SYSTEM dets
  (* Version 1.0, 2023-01-24, obotnar *)
  APPLICATION detsApp
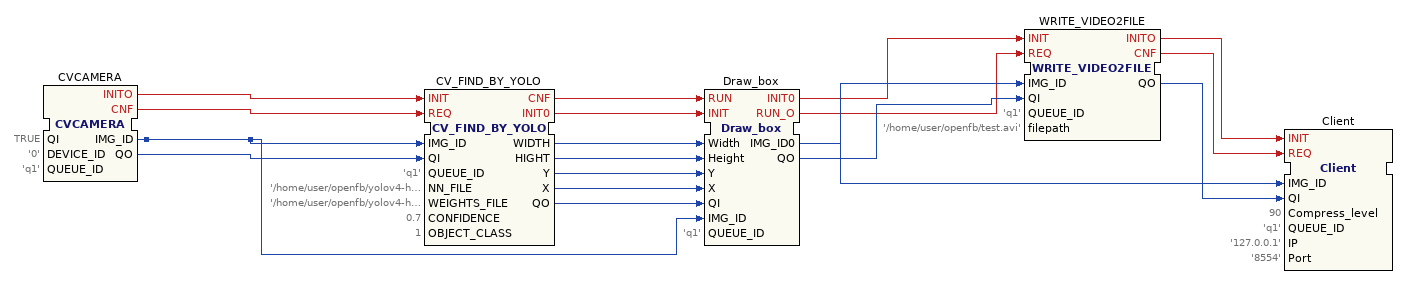
    FBS
      CV_FIND_BY_YOLO : CV_FIND_BY_YOLO(QUEUE_ID := 'q1', NN_FILE := '/home/user/openfb/yolov4-head-tiny-416.cfg', WEIGHTS_FILE := '/home/user/openfb/yolov4-head-tiny-416.weights', CONFIDENCE := 0.7, OBJECT_CLASS := 1);
      Draw_box : Draw_box(QUEUE_ID := 'q1');
      WRITE_VIDEO2FILE : WRITE_VIDEO2FILE(QUEUE_ID := 'q1', filepath := '/home/user/openfb/test.avi');
      Client : Client(Compress_level := 90, QUEUE_ID := 'q1', IP := '127.0.0.1', Port := '8554');
      CVCAMERA : CVCAMERA(QI := TRUE, DEVICE_ID := '0', QUEUE_ID := 'q1');
    END_FBS
    EVENT_CONNECTIONS
      CV_FIND_BY_YOLO.CNF TO Draw_box.RUN;
      CV_FIND_BY_YOLO.INIT0 TO Draw_box.INIT;
      Draw_box.INIT0 TO WRITE_VIDEO2FILE.INIT;
      Draw_box.RUN_O TO WRITE_VIDEO2FILE.REQ;
      WRITE_VIDEO2FILE.INITO TO Client.INIT;
      WRITE_VIDEO2FILE.CNF TO Client.REQ;
      CVCAMERA.INITO TO CV_FIND_BY_YOLO.INIT;
      CVCAMERA.CNF TO CV_FIND_BY_YOLO.REQ;
    END_CONNECTIONS
    DATA_CONNECTIONS
      CV_FIND_BY_YOLO.WIDTH TO Draw_box.Width;
      CV_FIND_BY_YOLO.HIGHT TO Draw_box.Height;
      CV_FIND_BY_YOLO.Y TO Draw_box.Y;
      CV_FIND_BY_YOLO.X TO Draw_box.X;
      CV_FIND_BY_YOLO.QO TO Draw_box.QI;
      Draw_box.IMG_ID0 TO WRITE_VIDEO2FILE.IMG_ID;
      Draw_box.QO TO WRITE_VIDEO2FILE.QI;
      Draw_box.IMG_ID0 TO Client.IMG_ID;
      WRITE_VIDEO2FILE.QO TO Client.QI;
      CVCAMERA.IMG_ID TO Draw_box.IMG_ID;
      CVCAMERA.IMG_ID TO CV_FIND_BY_YOLO.IMG_ID;
      CVCAMERA.QO TO CV_FIND_BY_YOLO.QI;
    END_CONNECTIONS
  END_APPLICATION
  DEVICE FORTE_PC : FORTE_PC(MGR_ID := "10.5.20.122:61499" (* Device manager socket ID *))
    {SET_ATTRIBUTE(Profile, HOLOBLOC)}
    RESOURCE EMB_RES : 
    END_RESOURCE
  END_DEVICE
  MAPPINGS
    detsApp.CV_FIND_BY_YOLO ON FORTE_PC.EMB_RES;
    detsApp.Draw_box ON FORTE_PC.EMB_RES;
    detsApp.WRITE_VIDEO2FILE ON FORTE_PC.EMB_RES;
    detsApp.Client ON FORTE_PC.EMB_RES;
    detsApp.CVCAMERA ON FORTE_PC.EMB_RES;
  END_MAPPINGS
  SEGMENTS
    Ethernet : Ethernet;
  END_SEGMENTS
  LINKS
    FORTE_PC => Ethernet;
  END_LINKS
END_SYSTEM
